TEXTLIST SafetyConfigTabsTextList
  0 = 'General'
  1 = 'Sound alert - bypassing'
  2 = 'LED alert - bypassing permanently'
  3 = 'Sound alert - doors opening when entering'
  4 = 'Sound alert - doors opening when leaving'
  5 = 'Sound alert - leaving when doors closed'
  6 = 'Sound alert - leavingwhen doors still open'
  7 = 'LED alert - doors are open'
   = ''
END_TEXTLIST

(* stored: Version 1.1.0.1, ProductVersion 3.1.4018.5
   TextList SafetyConfigTabsTextList: Id {9ae1ce35-ce16-435a-af60-63db3af4b4b5} *)
